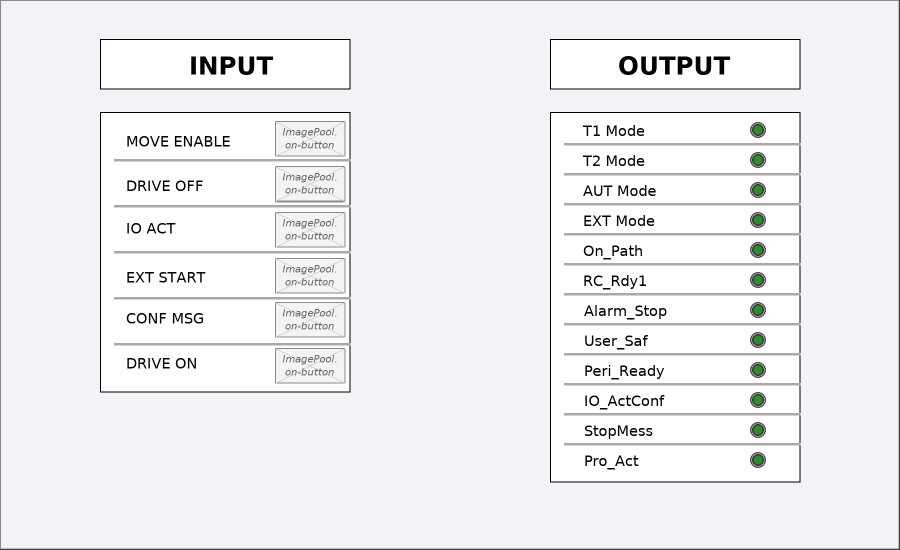
VISUALIZATION KUKA_IO_CONTENT  // 900x550
    Rectangle (0,0 900x550)
    RoundedRectangle (100,39 250x50)
    Rectangle (172,51 118x30), "INPUT"
    Group (100,112 250x280)
        RoundedRectangle (0,0 250x280)
        RoundedRectangle (23,21 153x17), "MOVE ENABLE"
        RoundedRectangle (23,65 92x18), "DRIVE OFF"
        RoundedRectangle (23,100 92x33), "IO ACT"
        RoundedRectangle (23,149 92x33), "EXT START"
        RoundedRectangle (23,190 92x33), "CONF MSG"
        RoundedRectangle (23,235 92x33), "DRIVE ON"
        Image (175,9 70x35), invisible if: IO_KUKA.bMove_enable, image: ImagePool.off-button
            OnMouseClick: toggle IO_HMI.bMove_enable
        Image (175,9 70x35), invisible if: NOT IO_KUKA.bMove_enable, image: ImagePool.on-button
            OnMouseClick: toggle IO_HMI.bMove_enable
        Image (175,55 70x35), invisible if: IO_KUKA.bDrive_off, image: ImagePool.off-button
            OnMouseClick: toggle IO_HMI.bDrive_off
        Image (175,54 70x35), invisible if: NOT IO_KUKA.bDrive_off, image: ImagePool.on-button
            OnMouseClick: toggle IO_HMI.bDrive_off
        Image (175,100 70x35), invisible if: IO_KUKA.bIO_Act, image: ImagePool.off-button
            OnMouseClick: toggle IO_HMI.bIO_Act
        Image (175,100 70x35), invisible if: NOT IO_KUKA.bIO_Act, image: ImagePool.on-button
            OnMouseClick: toggle IO_HMI.bIO_Act
        Image (175,146 70x35), invisible if: IO_KUKA.bExt_start, image: ImagePool.off-button
            OnMouseClick: toggle IO_HMI.bExt_start
        Image (175,146 70x35), invisible if: NOT IO_KUKA.bExt_start, image: ImagePool.on-button
            OnMouseClick: toggle IO_HMI.bExt_start
        Image (175,190 70x35), invisible if: IO_KUKA.bConf_msg, image: ImagePool.off-button
            OnMouseClick: toggle IO_HMI.bConf_msg
        Image (175,190 70x35), invisible if: NOT IO_KUKA.bConf_msg, image: ImagePool.on-button
            OnMouseClick: toggle IO_HMI.bConf_msg
        Image (175,236 70x35), invisible if: IO_KUKA.bDrive_on, image: ImagePool.off-button
            OnMouseClick: toggle IO_HMI.bDrive_on
        Image (175,236 70x35), invisible if: NOT IO_KUKA.bDrive_on, image: ImagePool.on-button
            OnMouseClick: toggle IO_HMI.bDrive_on
        Rectangle (14,47 236x2)
        Rectangle (14,93 236x2)
        Rectangle (14,139 236x2)
        Rectangle (14,185 236x2)
        Rectangle (14,231 236x2)
    Group (550,112 250x370)
        RoundedRectangle (0,0 250x370)
        Rectangle (30,4 118x30), "T1 Mode"
        Rectangle (30,34 118x30), "T2 Mode"
        Rectangle (30,64 118x30), "AUT Mode"
        Rectangle (30,94 118x30), "EXT Mode"
        Rectangle (30,124 118x30), "On_Path"
        Rectangle (30,154 118x30), "RC_Rdy1"
        Rectangle (31,184 118x30), "Alarm_Stop"
        Rectangle (31,214 118x30), "User_Saf"
        Rectangle (31,244 118x30), "Peri_Ready"
        Rectangle (31,274 118x30), "IO_ActConf"
        Rectangle (31,304 118x30), "StopMess"
        Rectangle (31,334 118x30), "Pro_Act"
        Lamp1 (199,9 18x18), variable: IO_KUKA.bT1_mode, style: Lamp-Lamp1-Green
        Lamp1 (199,39 18x18), variable: IO_KUKA.bT2_mode, style: Lamp-Lamp1-Green
        Lamp1 (199,69 18x18), variable: IO_KUKA.bAUT_mode, style: Lamp-Lamp1-Green
        Lamp1 (199,99 18x18), variable: IO_KUKA.bEXT_mode, style: Lamp-Lamp1-Green
        Lamp1 (199,129 18x18), variable: IO_KUKA.bOn_path, style: Lamp-Lamp1-Green
        Lamp1 (199,159 18x18), variable: IO_KUKA.bRC_ready, style: Lamp-Lamp1-Green
        Lamp1 (199,189 18x18), variable: IO_KUKA.bAlarm_stop, style: Lamp-Lamp1-Green
        Lamp1 (199,219 18x18), variable: IO_KUKA.bUser_safety, style: Lamp-Lamp1-Green
        Lamp1 (199,249 18x18), variable: IO_KUKA.bPeri_ready, style: Lamp-Lamp1-Green
        Lamp1 (199,279 18x18), variable: IO_KUKA.bIO_ActConf, style: Lamp-Lamp1-Green
        Lamp1 (199,309 18x18), variable: IO_KUKA.bStopmess, style: Lamp-Lamp1-Green
        Lamp1 (199,339 18x18), variable: IO_KUKA.bPro_act, style: Lamp-Lamp1-Green
        Rectangle (14,31 236x2)
        Rectangle (14,61 236x2)
        Rectangle (14,211 236x2)
        Rectangle (14,241 236x2)
        Rectangle (14,271 236x2)
        Rectangle (14,181 236x2)
        Rectangle (14,151 236x2)
        Rectangle (14,121 236x2)
        Rectangle (14,91 236x2)
        Rectangle (14,301 236x2)
        Rectangle (14,331 236x2)
    RoundedRectangle (550,39 250x50)
    Rectangle (615,51 118x30), "OUTPUT"
END_VISUALIZATION

(* stored: Version 1.1.0.1, ProductVersion 3.1.4024.12
   Visu KUKA_IO_CONTENT: Id {ca894096-c391-420e-a42c-cdb312d3993d} *)
